// TIA Portal V20 export
TYPE "LKinCtrl_Utilities_typeChangeSelectionConfiguration"
// stored: Access Published
   STRUCT
      noSelection { ExternalAccessible := 'False'; ExternalVisible := 'False'; ExternalWritable := 'False'} : Bool;   // TRUE: Select nothing.
      firstSelectedIndex { ExternalAccessible := 'False'; ExternalVisible := 'False'; ExternalWritable := 'False'} : DInt;   // First selected index., if noSelection = FALSE.
      lastSelectedIndex { ExternalAccessible := 'False'; ExternalVisible := 'False'; ExternalWritable := 'False'} : DInt;   // Last selected index, if noSelection = FALSE and multiSelection enabled.
   END_STRUCT;
END_TYPE
